TYPE ST_DiscreteValveState :
STRUCT
	bValveIsOpen : BOOL;
END_STRUCT
END_TYPE

(* stored: Version 1.1.0.1, ProductVersion 3.1.4024.9
   DUT ST_DiscreteValveState: Id {6e7181a3-d3f3-4c12-8906-3e401b341bd3} *)
